// Mitsubishi GX Works2 project: group_8 working_toSubmit   PLC: FX3G

// global labels: Global1
VAR_GLOBAL
  SW_7_StartDay AT X007 : BOOL;
  Li_7_Day AT M5 : BOOL;
  SW_11_emergency AT X011 : BOOL;
  Supply_end AT M1 : BOOL;
  Shmarim_Input_Amount AT D1148 : REAL;
  Letet_Input_Amount AT D1195 : REAL;
  Reg_Shmarimg_Amount AT D1150 : REAL;
  Reg_Letet_Amount AT D1200 : REAL;
  Reg_Kshut_Amount AT D1250 : REAL;
  Beer_Input AT D8280 : INT;
  Final_Beer_Type AT D1155 : REAL;
END_VAR
VAR_GLOBAL CONSTANT
  const_5 : REAL := 5;
END_VAR
VAR_GLOBAL
  Pilsner AT M2 : BOOL;
  Lager AT M3 : BOOL;
END_VAR
VAR_GLOBAL CONSTANT
  const_400 : INT := 400;
END_VAR
VAR_GLOBAL
  Kshut_Input_Amount AT D1245 : REAL;
END_VAR
VAR_GLOBAL CONSTANT
  const_10 : REAL := 10;
  Const_6 : REAL := 6;
END_VAR
VAR_GLOBAL
  Check_Supply AT M4 : BOOL;
END_VAR
VAR_GLOBAL CONSTANT
  const_150 : REAL := 150;
  const_12 : REAL := 12;
  Const_60 : REAL := 60;
  const_120 : REAL := 120;
  Const_53 : REAL := 53;
END_VAR
VAR_GLOBAL
  Timer_brew4 AT TC1 : BOOL;
END_VAR
VAR_GLOBAL CONSTANT
  For_sec_brew : INT := K40;
END_VAR
VAR_GLOBAL
  Timer_brew_finish AT TS1 : BOOL;
  Start_brew AT X001 : BOOL;
  is_brew AT Y001 : BOOL;
  lamp_start_day AT Y007 : BOOL;
  Start_fermentation AT X005 : BOOL;
  stop_pilzner_timer AT TS2 : BOOL;
  timer_bliking_pilsner AT TC2 : BOOL;
END_VAR
VAR_GLOBAL CONSTANT
  pilzner_bilking_time : INT := 40;
END_VAR
VAR_GLOBAL
  timer_bliking_lager AT TC3 : BOOL;
END_VAR
VAR_GLOBAL CONSTANT
  Lager_bilking_timer : INT := 30;
END_VAR
VAR_GLOBAL
  stop_lager_timer AT TS3 : BOOL;
  end_timer_pilzner AT M7 : BOOL;
  end_timer_lager AT M6 : BOOL;
  lamp_y3 AT Y003 : BOOL;
END_VAR
VAR_GLOBAL CONSTANT
  bliking_timer_y3 : INT := 5;
END_VAR
VAR_GLOBAL
  bliking_y4 AT TC5 : BOOL;
END_VAR
VAR_GLOBAL CONSTANT
  bliking_timer_y4 : INT := 5;
END_VAR
VAR_GLOBAL
  stop_bliking_y3 AT TS4 : BOOL;
  indicator_bliking_1 AT M0 : BOOL;
  bliking_y3 AT TC4 : BOOL;
  lamp_y4 AT Y004 : BOOL;
  stop_bliking_y4 AT TS5 : BOOL;
  Start_Botteling AT X002 : BOOL;
  Lamp_y2 AT Y002 : BOOL;
  first_bottling AT X000 : BOOL;
END_VAR
VAR_GLOBAL CONSTANT
  couter_six_beers : INT := 6;
  const_1 : INT := 1;
END_VAR
VAR_GLOBAL
  current_counter_beers AT CN1 : INT;
END_VAR
VAR_GLOBAL CONSTANT
  const_5_word : INT := 5;
END_VAR
VAR_GLOBAL
  Pilsner_help AT M50 : BOOL;
  Lager_help AT M51 : BOOL;
END_VAR
VAR_GLOBAL CONSTANT
  ADD_Package : REAL := 1;
END_VAR
VAR_GLOBAL
  Amount_packages AT D1160 : REAL;
END_VAR
VAR_GLOBAL CONSTANT
  MUL40 : REAL := 40;
END_VAR
VAR_GLOBAL
  OutputMul AT D1170 : REAL;
  output AT D8282 : INT;
  M_add_Package AT M98 : BOOL;
  not_enough_for_pilsner AT M60 : BOOL;
  not_enough_for_lagger AT M61 : BOOL;
  end_day AT M10 : BOOL;
  raw_materialsl_brew AT D1190 : REAL;
END_VAR
VAR_GLOBAL CONSTANT
  const_222_lager_braw : REAL := 222;
  const_179_Pilsner_braw : REAL := 179;
END_VAR
VAR_GLOBAL
  help_not_enough_for_pilsner AT M65 : BOOL;
  help_not_enough_for_lagger AT M67 : BOOL;
  finish_six AT CS1 : BOOL;
  done_six AT CC1 : BOOL;
  raw_materialsl_ferm AT D1165 : REAL;
END_VAR

// task Task_01 (event TRUE, interval 0, priority 31): POU_01

PROGRAM POU_01
(* structured ladder/FBD written out as ST: instructions are called as NAME(EN, inputs, outputs); _pN, _eN, _tN stand for wires *)
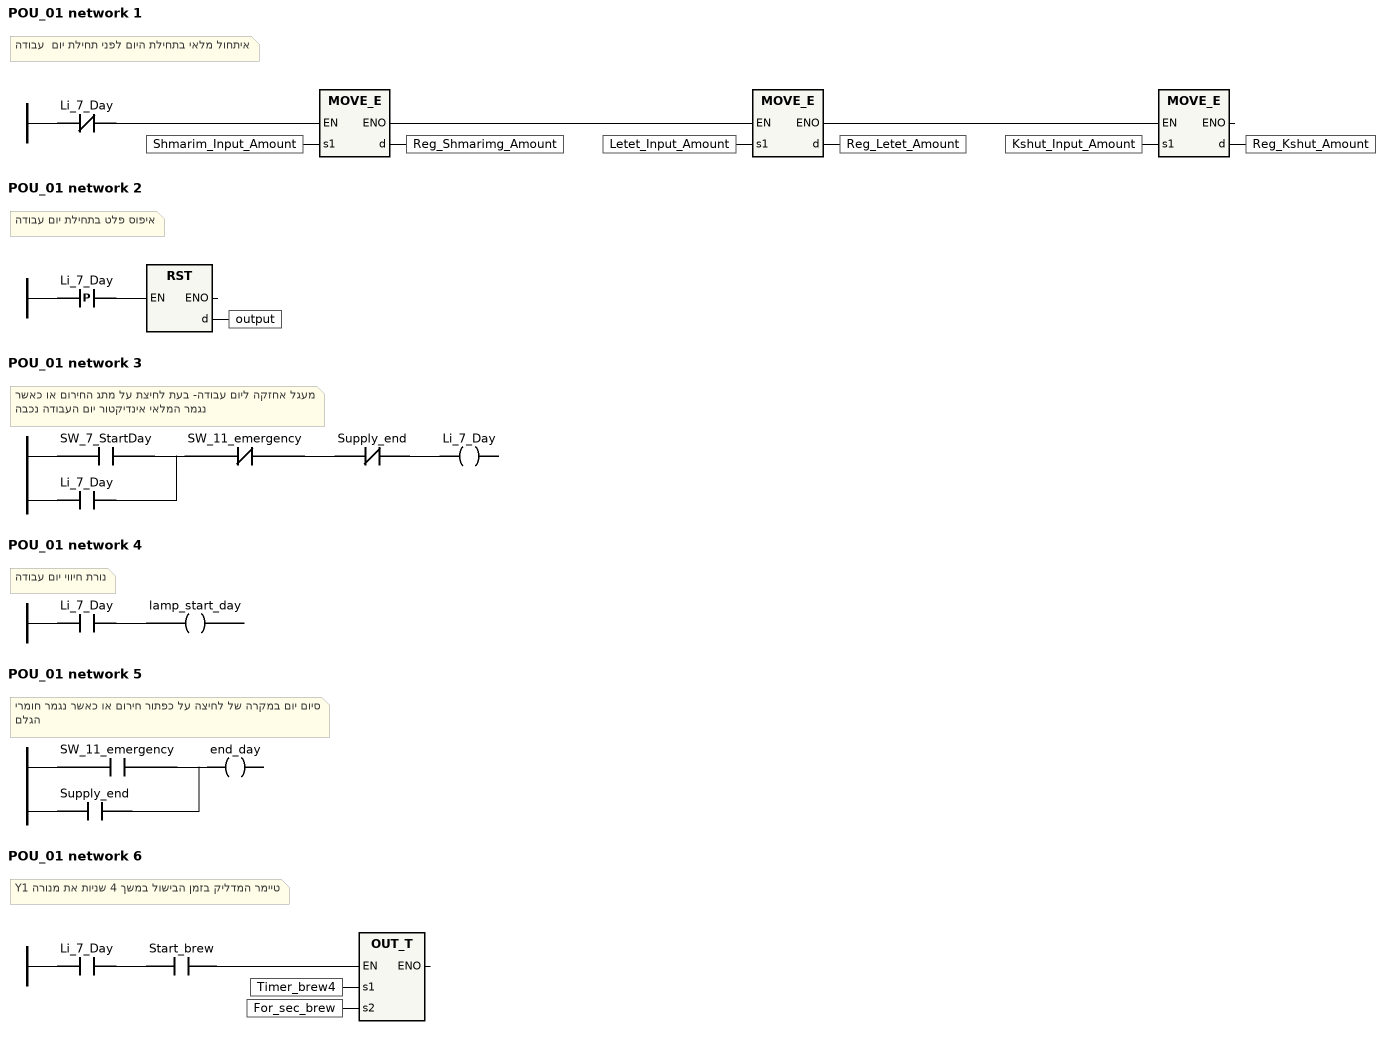
(* network 1 *)
(* איתחול מלאי בתחילת היום לפני תחילת יום  עבודה *)
_e1 := MOVE_E(NOT Li_7_Day, Shmarim_Input_Amount, Reg_Shmarimg_Amount);
_e2 := MOVE_E(_e1, Letet_Input_Amount, Reg_Letet_Amount);
MOVE_E(_e2, Kshut_Input_Amount, Reg_Kshut_Amount);
(* network 2 *)
(* איפוס פלט בתחילת יום עבודה *)
RST(LDP(TRUE, Li_7_Day), output);
(* network 3 *)
(* מעגל אחזקה ליום עבודה- בעת לחיצת על מתג החירום או כאשר נגמר המלאי אינדיקטור יום העבודה נכבה *)
Li_7_Day := ((SW_7_StartDay OR Li_7_Day) AND NOT SW_11_emergency) AND NOT Supply_end;
(* network 4 *)
(* נורת חיווי יום עבודה *)
lamp_start_day := Li_7_Day;
(* network 5 *)
(* סיום יום במקרה של לחיצה על כפתור חירום או כאשר נגמר חומרי הגלם *)
end_day := SW_11_emergency OR Supply_end;
(* network 6 *)
(* טיימר המדליק בזמן הבישול במשך 4 שניות את מנורה Y1 *)
OUT_T(Li_7_Day AND Start_brew, Timer_brew4, For_sec_brew);
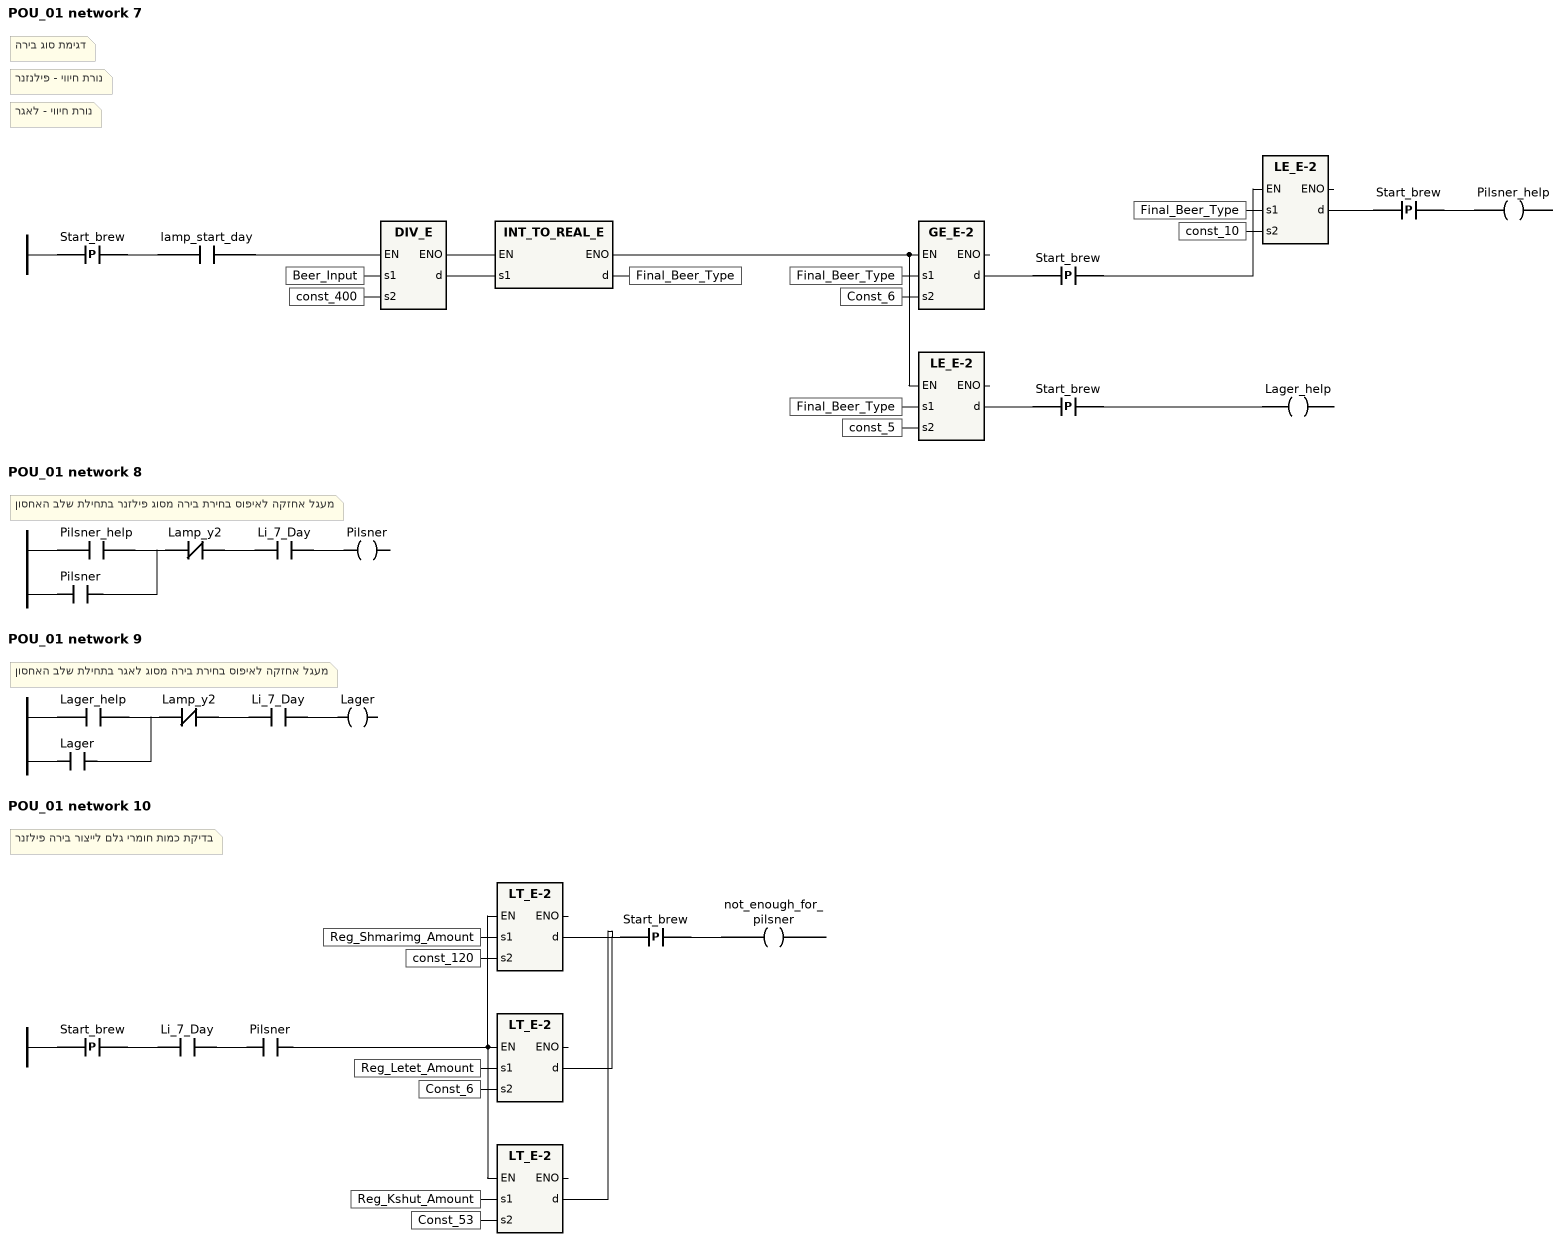
(* network 7 *)
(* דגימת סוג בירה *)
(* נורת חיווי - פילנזנר *)
(* נורת חיווי - לאגר *)
_e2 := DIV_E(LDP(TRUE, Start_brew) AND lamp_start_day, Beer_Input, const_400, _t1);
_e3 := INT_TO_REAL_E(_e2, _t1, Final_Beer_Type);
GE_E(_e3, Final_Beer_Type, Const_6, _t4);
LE_E(_t4 AND LDP(TRUE, Start_brew), Final_Beer_Type, const_10, _t5);
Pilsner_help := _t5 AND LDP(TRUE, Start_brew);
LE_E(_e3, Final_Beer_Type, const_5, _t6);
Lager_help := _t6 AND LDP(TRUE, Start_brew);
(* network 8 *)
(* מעגל אחזקה לאיפוס בחירת בירה מסוג פילזנר בתחילת שלב האחסון *)
Pilsner := ((Pilsner_help OR Pilsner) AND NOT Lamp_y2) AND Li_7_Day;
(* network 9 *)
(* מעגל אחזקה לאיפוס בחירת בירה מסוג לאגר בתחילת שלב האחסון *)
Lager := ((Lager_help OR Lager) AND NOT Lamp_y2) AND Li_7_Day;
(* network 10 *)
(* בדיקת כמות חומרי גלם לייצור בירה פילזנר *)
_p1 := LDP(TRUE, Start_brew) AND Li_7_Day AND Pilsner;
LT_E(_p1, Reg_Shmarimg_Amount, const_120, _t2);
LT_E(_p1, Reg_Letet_Amount, Const_6, _t3);
LT_E(_p1, Reg_Kshut_Amount, Const_53, _t4);
not_enough_for_pilsner := (_t2 OR _t3 OR _t4) AND LDP(TRUE, Start_brew);
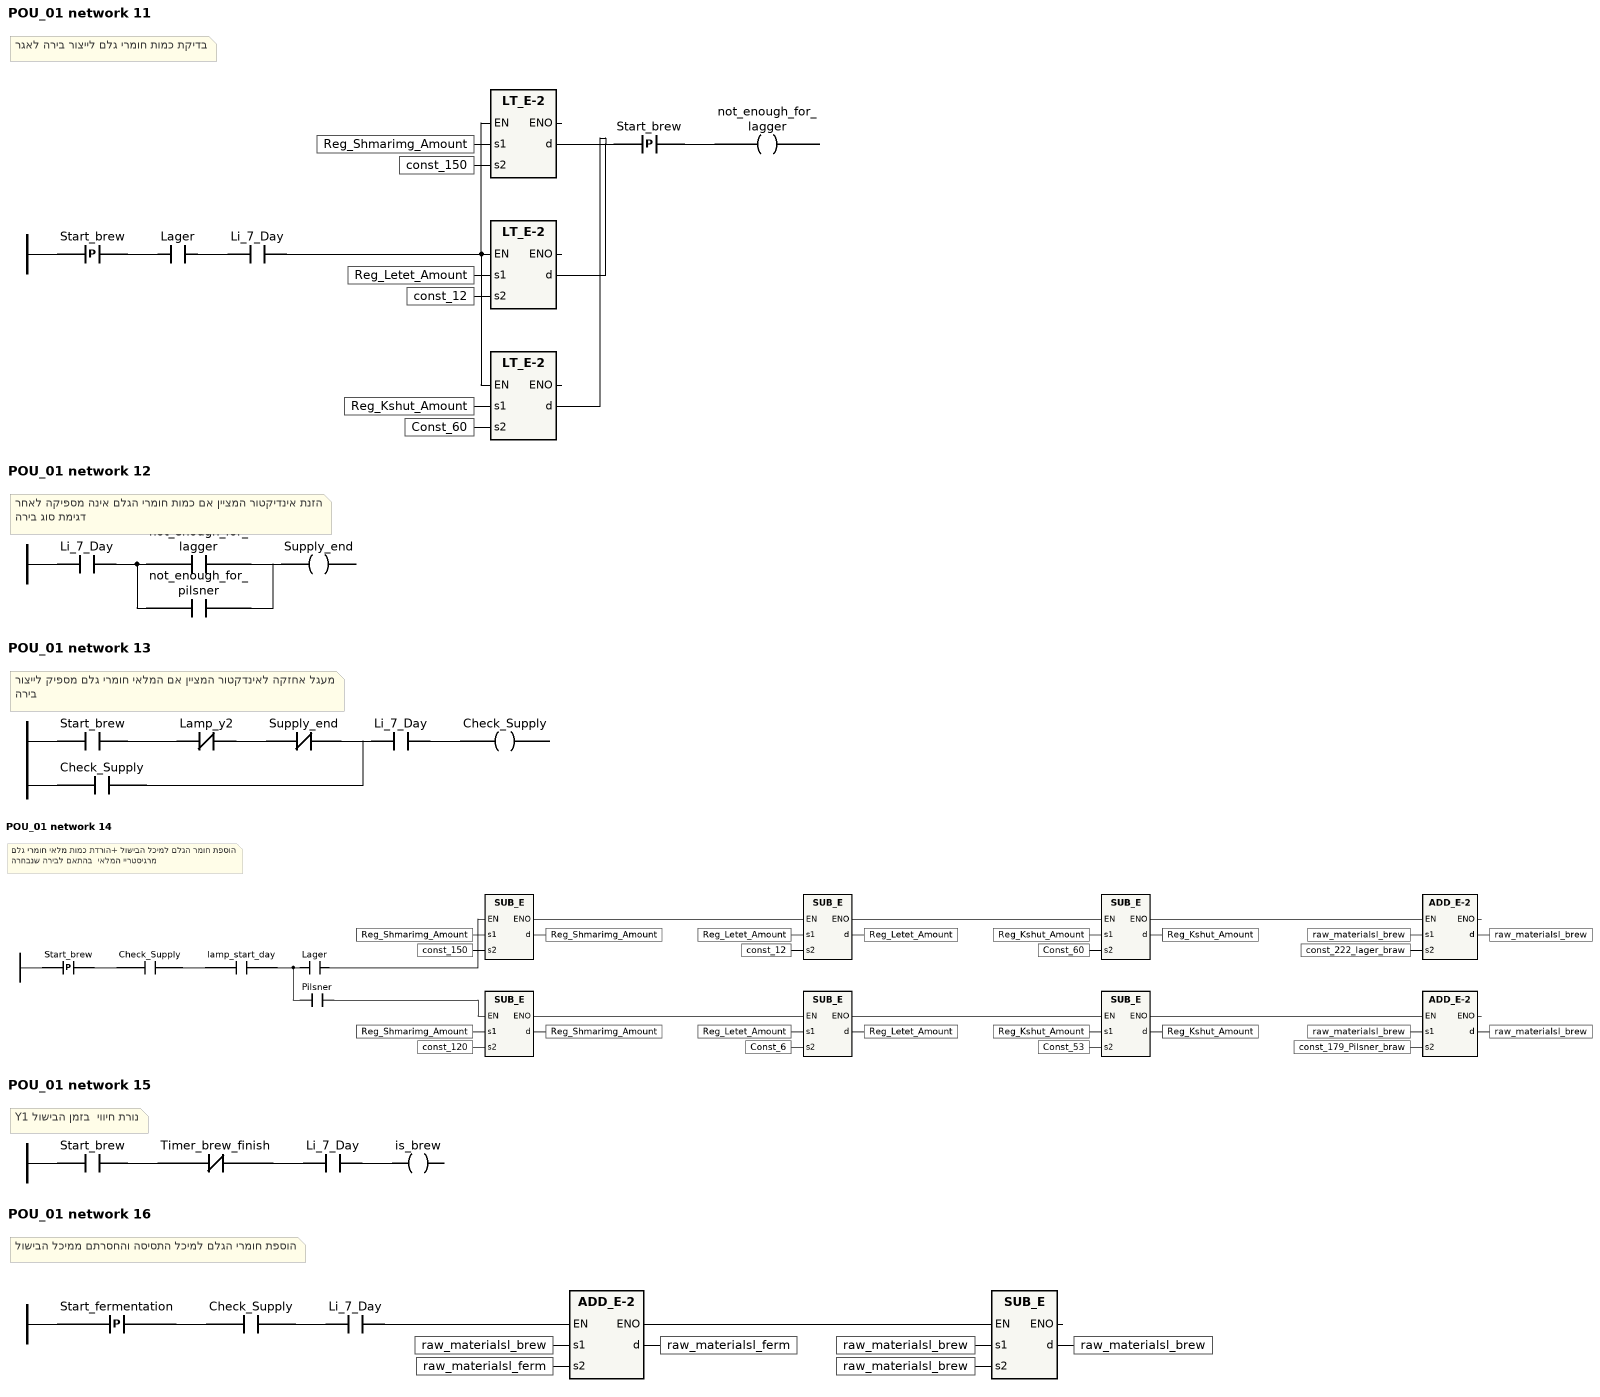
(* network 11 *)
(* בדיקת כמות חומרי גלם לייצור בירה לאגר *)
_p1 := LDP(TRUE, Start_brew) AND Lager AND Li_7_Day;
LT_E(_p1, Reg_Shmarimg_Amount, const_150, _t2);
LT_E(_p1, Reg_Letet_Amount, const_12, _t3);
LT_E(_p1, Reg_Kshut_Amount, Const_60, _t4);
not_enough_for_lagger := (_t2 OR _t3 OR _t4) AND LDP(TRUE, Start_brew);
(* network 12 *)
(* הזנת אינדיקטור המציין אם כמות חומרי הגלם אינה מספיקה לאחר דגימת סוג בירה *)
Supply_end := (Li_7_Day AND not_enough_for_lagger) OR (Li_7_Day AND not_enough_for_pilsner);
(* network 13 *)
(* מעגל אחזקה לאינדקטור המציין אם המלאי חומרי גלם מספיק לייצור בירה *)
Check_Supply := ((Start_brew AND NOT Lamp_y2 AND NOT Supply_end) OR Check_Supply) AND Li_7_Day;
(* network 14 *)
(* הוספת חומר הגלם למיכל הבישול +הורדת כמות מלאי חומרי גלם מרגיסטריי המלאי  בהתאם לבירה שנבחרה *)
_p1 := LDP(TRUE, Start_brew) AND Check_Supply AND lamp_start_day;
_e2 := SUB_E(_p1 AND Lager, Reg_Shmarimg_Amount, const_150, Reg_Shmarimg_Amount);
_e3 := SUB_E(_e2, Reg_Letet_Amount, const_12, Reg_Letet_Amount);
_e4 := SUB_E(_e3, Reg_Kshut_Amount, Const_60, Reg_Kshut_Amount);
ADD_E(_e4, raw_materialsl_brew, const_222_lager_braw, raw_materialsl_brew);
_e5 := SUB_E(_p1 AND Pilsner, Reg_Shmarimg_Amount, const_120, Reg_Shmarimg_Amount);
_e6 := SUB_E(_e5, Reg_Letet_Amount, Const_6, Reg_Letet_Amount);
_e7 := SUB_E(_e6, Reg_Kshut_Amount, Const_53, Reg_Kshut_Amount);
ADD_E(_e7, raw_materialsl_brew, const_179_Pilsner_braw, raw_materialsl_brew);
(* network 15 *)
(* נורת חיווי  בזמן הבישול Y1 *)
is_brew := Start_brew AND NOT Timer_brew_finish AND Li_7_Day;
(* network 16 *)
(* הוספת חומרי הגלם למיכל התסיסה והחסרתם ממיכל הבישול *)
_e1 := ADD_E(LDP(TRUE, Start_fermentation) AND Check_Supply AND Li_7_Day, raw_materialsl_brew, raw_materialsl_ferm, raw_materialsl_ferm);
SUB_E(_e1, raw_materialsl_brew, raw_materialsl_brew, raw_materialsl_brew);
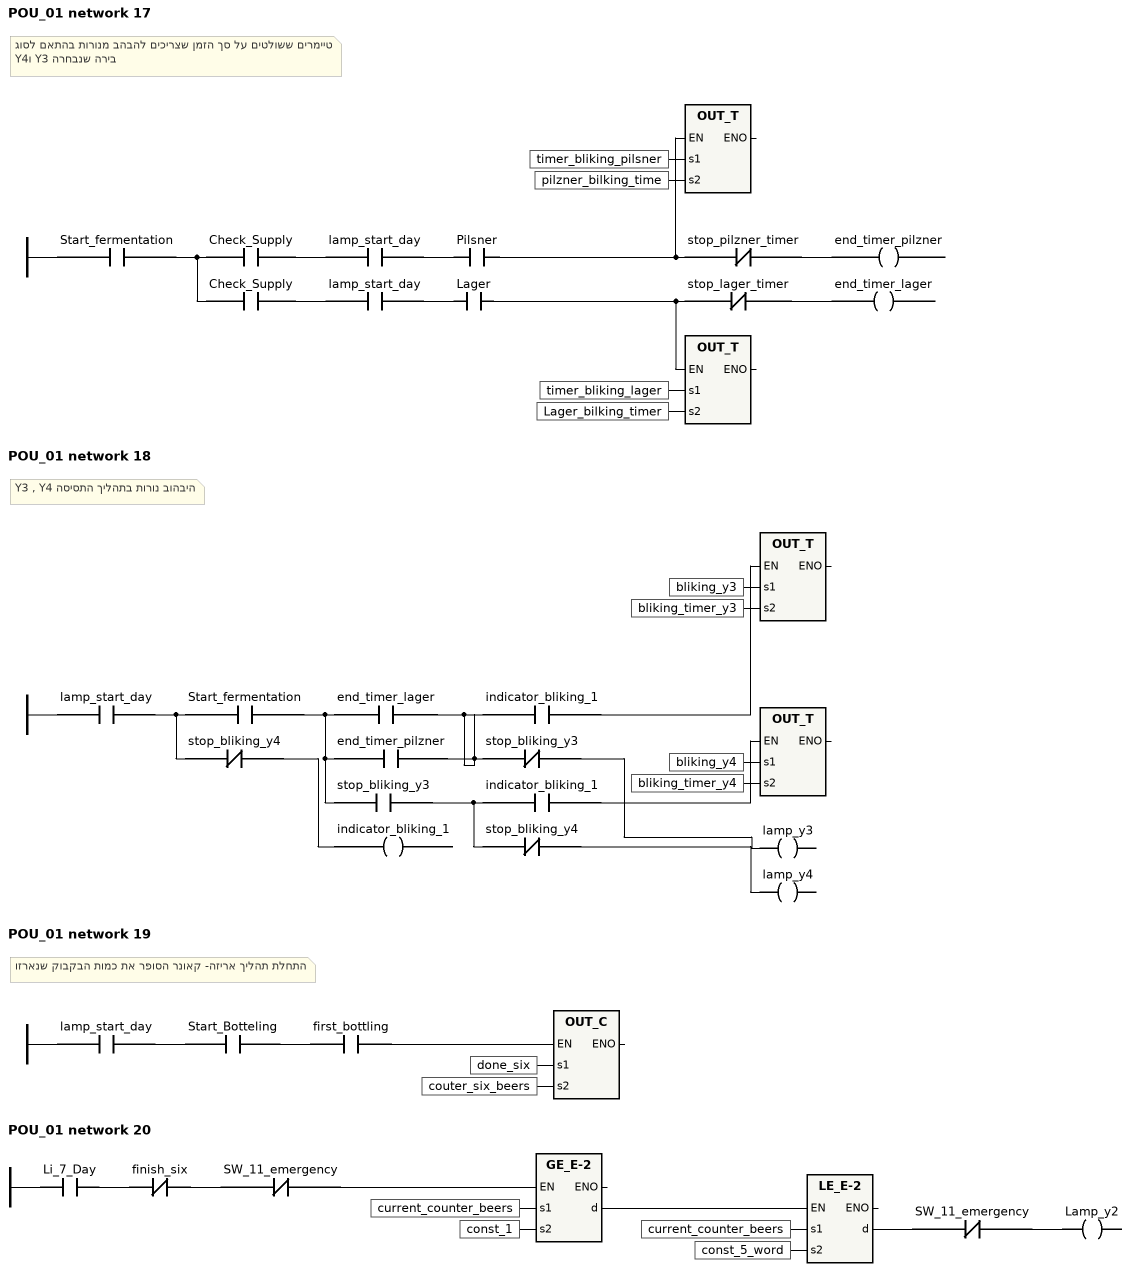
(* network 17 *)
(* טיימרים ששולטים על סך הזמן שצריכים להבהב מנורות בהתאם לסוג בירה שנבחרה Y3 וY4 *)
_p1 := Start_fermentation AND Check_Supply AND lamp_start_day AND Pilsner;
OUT_T(_p1, timer_bliking_pilsner, pilzner_bilking_time);
end_timer_pilzner := _p1 AND NOT stop_pilzner_timer;
_p2 := Start_fermentation AND Check_Supply AND lamp_start_day AND Lager;
OUT_T(_p2, timer_bliking_lager, Lager_bilking_timer);
end_timer_lager := _p2 AND NOT stop_lager_timer;
(* network 18 *)
(* היבהוב נורות בתהליך התסיסה Y3 , Y4 *)
_p1 := lamp_start_day AND Start_fermentation;
_p2 := (_p1 AND end_timer_lager) OR (_p1 AND end_timer_pilzner);
OUT_T(_p2 AND indicator_bliking_1, bliking_y3, bliking_timer_y3);
lamp_y3 := _p2 AND NOT stop_bliking_y3;
_p3 := _p1 AND stop_bliking_y3;
OUT_T(_p3 AND indicator_bliking_1, bliking_y4, bliking_timer_y4);
lamp_y4 := _p3 AND NOT stop_bliking_y4;
indicator_bliking_1 := lamp_start_day AND NOT stop_bliking_y4;
(* network 19 *)
(* התחלת תהליך אריזה- קאונר הסופר את כמות הבקבוק שנארזו *)
OUT_C(lamp_start_day AND Start_Botteling AND first_bottling, done_six, couter_six_beers);
(* network 20 *)
GE_E(Li_7_Day AND NOT finish_six AND NOT SW_11_emergency, current_counter_beers, const_1, _t1);
LE_E(_t1, current_counter_beers, const_5_word, _t2);
Lamp_y2 := _t2 AND NOT SW_11_emergency;
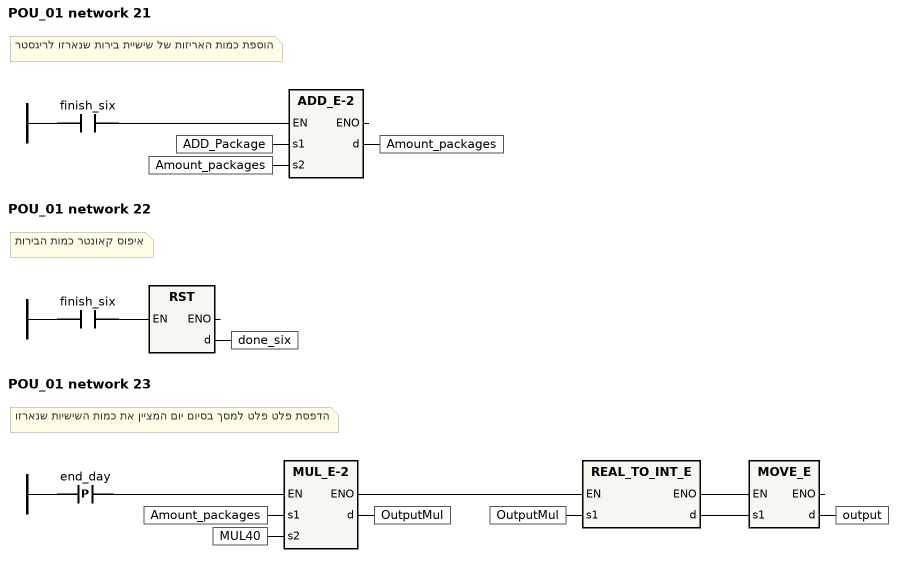
(* network 21 *)
(* הוספת כמות האריזות של שישיית בירות שנארזו לריגסטר *)
ADD_E(finish_six, ADD_Package, Amount_packages, Amount_packages);
(* network 22 *)
(* איפוס קאונטר כמות הבירות *)
RST(finish_six, done_six);
(* network 23 *)
(* הדפסת פלט פלט למסך בסיום יום המציין את כמות השישיות שנארזו *)
_e1 := MUL_E(LDP(TRUE, end_day), Amount_packages, MUL40, OutputMul);
_e3 := REAL_TO_INT_E(_e1, OutputMul, _t2);
MOVE_E(_e3, _t2, output);
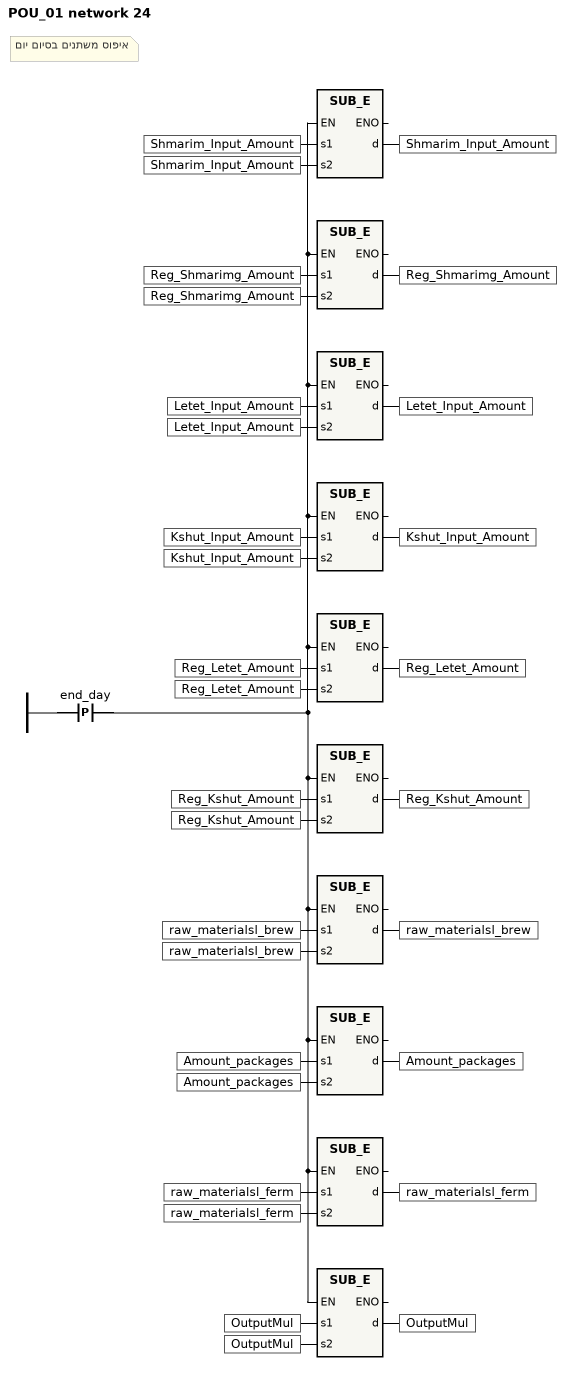
(* network 24 *)
(* איפוס משתנים בסיום יום *)
_p1 := LDP(TRUE, end_day);
SUB_E(_p1, Shmarim_Input_Amount, Shmarim_Input_Amount, Shmarim_Input_Amount);
SUB_E(_p1, Reg_Shmarimg_Amount, Reg_Shmarimg_Amount, Reg_Shmarimg_Amount);
SUB_E(_p1, Letet_Input_Amount, Letet_Input_Amount, Letet_Input_Amount);
SUB_E(_p1, Kshut_Input_Amount, Kshut_Input_Amount, Kshut_Input_Amount);
SUB_E(_p1, Reg_Letet_Amount, Reg_Letet_Amount, Reg_Letet_Amount);
SUB_E(_p1, Reg_Kshut_Amount, Reg_Kshut_Amount, Reg_Kshut_Amount);
SUB_E(_p1, raw_materialsl_brew, raw_materialsl_brew, raw_materialsl_brew);
SUB_E(_p1, Amount_packages, Amount_packages, Amount_packages);
SUB_E(_p1, raw_materialsl_ferm, raw_materialsl_ferm, raw_materialsl_ferm);
SUB_E(_p1, OutputMul, OutputMul, OutputMul);
END_PROGRAM
